# EPICS substitutions: ATCACommonApp/Db/StreamShort.substitutions
file "streamWf.db"  {
    pattern {      PORT,   DEVICE,    WIDTH,  N,   TYPE,                DTYP,      FTVL,       NELM,    TSE      }
            { "$(PORT)", "$(DEV)",  "Int16", 0, "SHORT", "asynInt16ArrayOut",   "SHORT",  "$(NELM)", "$(TSE)"    }
            { "$(PORT)", "$(DEV)",  "Int16", 1, "SHORT", "asynInt16ArrayOut",   "SHORT",  "$(NELM)", "$(TSE)"    }
            { "$(PORT)", "$(DEV)",  "Int16", 2, "SHORT", "asynInt16ArrayOut",   "SHORT",  "$(NELM)", "$(TSE)"    }
            { "$(PORT)", "$(DEV)",  "Int16", 3, "SHORT", "asynInt16ArrayOut",   "SHORT",  "$(NELM)", "$(TSE)"    }

}
